// TIA Portal V18 export
DATA_BLOCK "PLC_2_Send_DB"   // DB23
{ S7_Optimized_Access := 'TRUE' }
// stored: InstanceOfName TCON_IP_v4, OfSystemLibElement TCON_IP_v4, OfSystemLibVersion 1.0
"TCON_IP_v4"
   // VAR
   //    InterfaceId : HW_ANY := 64;
   //    ID : CONN_OUC := 2;
   //    ConnectionType : Byte;
   //    ActiveEstablished : Bool := true;
   //    RemoteAddress { S7_SetPoint := 'True'} : IP_V4;
   //    RemotePort : UInt := 502;
   //    LocalPort : UInt := 0;
   // END_VAR
BEGIN
   RemoteAddress.ADDR[1] := 192;
   RemoteAddress.ADDR[2] := 168;
   RemoteAddress.ADDR[3] := 6;
   RemoteAddress.ADDR[4] := 11;
END_DATA_BLOCK
